(* CODESYS project PLC_Program.project

Project tree, tasks and I/O mapping:
  Device : CODESYS Control Win V3, 3S - Smart Software Solutions GmbH, order no. 305021, version 3.5.11.30
    application Application
      libraries: Standard, * (System)
      task MainTask (cyclic, interval t#20ms, priority 1) calls PLC_PRG
      task VISU_TASK (cyclic, interval 100 ms, priority 31) calls VisuElems.Visu_Prg
      program PLC_PRG [LD]
      visualisation Visualization
      Symbols
  libraries: VisuSymbols, 3.5.10.0 (System)
  text list GlobalTextList
*)

// Device/Application/PLC_PRG
PROGRAM PLC_PRG
VAR
	// TAGS DOS MÓDULOS DE ENTRADA DIGITAL E SAÍDA DIGITAL
	I0: BYTE;
	Q0: BYTE;
	// TAG DOS BLOCOS DE MEMÓRIA
	M0: BYTE;
END_VAR

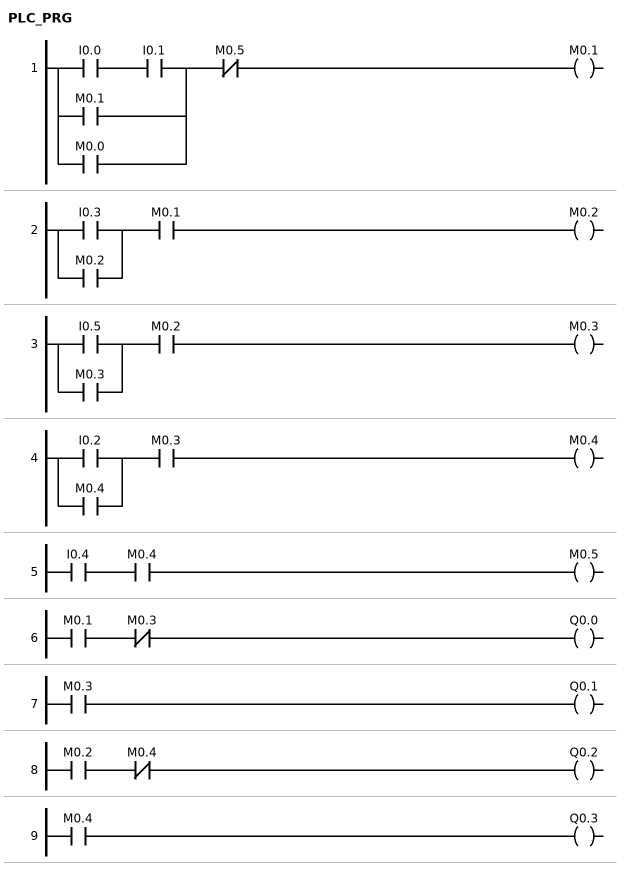
// NETWORK 1
M0.1 := (I0.0 AND I0.1 OR M0.1 OR M0.0) AND NOT M0.5;

// NETWORK 2
M0.2 := (I0.3 OR M0.2) AND M0.1;

// NETWORK 3
M0.3 := (I0.5 OR M0.3) AND M0.2;

// NETWORK 4
M0.4 := (I0.2 OR M0.4) AND M0.3;

// NETWORK 5
M0.5 := I0.4 AND M0.4;

// NETWORK 6
Q0.0 := M0.1 AND NOT M0.3;

// NETWORK 7
Q0.1 := M0.3;

// NETWORK 8
Q0.2 := M0.2 AND NOT M0.4;

// NETWORK 9
Q0.3 := M0.4;

END_PROGRAM

// Device/Application/Visualization
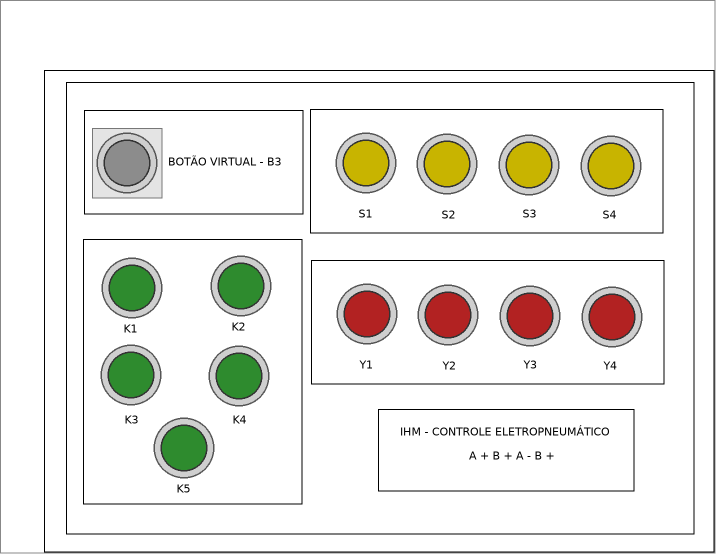
VISUALIZATION Visualization  // 716x554
    Rectangle (44,70 670x482)
    RoundedRectangle (66,82 628x452)
    RoundedRectangle (84,110 219x104)
    PushSwitch (92,128 70x70), variable: PLC_PRG.M0.0, behaviour: TOGGLE, style: Switch-PushSwitch-Gray
    Label (150,147 150x30), "BOTÃO VIRTUAL - B3"
    RoundedRectangle (310,109 353x124)
    Label (344,199 43x30), "S1"
    Lamp1 (331,128 70x70), variable: PLC_PRG.I0.2, style: Lamp-Lamp1-Yellow
    Lamp1 (412,129 70x70), variable: PLC_PRG.I0.3, style: Lamp-Lamp1-Yellow
    Lamp1 (494,130 70x70), variable: PLC_PRG.I0.4, style: Lamp-Lamp1-Yellow
    Lamp1 (576,131 70x70), variable: PLC_PRG.I0.5, style: Lamp-Lamp1-Yellow
    Label (427,200 43x30), "S2"
    Label (508,199 43x30), "S3"
    Label (588,200 43x30), "S4"
    RoundedRectangle (311,260 353x124)
    Label (345,350 43x30), "Y1"
    Lamp1 (332,279 70x70), variable: PLC_PRG.Q0.0, style: Lamp-Lamp1-Red
    Lamp1 (413,280 70x70), variable: PLC_PRG.Q0.1, style: Lamp-Lamp1-Red
    Lamp1 (495,281 70x70), variable: PLC_PRG.Q0.2, style: Lamp-Lamp1-Red
    Lamp1 (577,282 70x70), variable: PLC_PRG.Q0.3, style: Lamp-Lamp1-Red
    Label (428,351 43x30), "Y2"
    Label (509,350 43x30), "Y3"
    Label (589,351 43x30), "Y4"
    RoundedRectangle (83,239 219x265)
    Lamp1 (97,253 70x70), variable: PLC_PRG.M0.1, style: Lamp-Lamp1-Green
    Lamp1 (206,251 70x70), variable: PLC_PRG.M0.2, style: Lamp-Lamp1-Green
    Lamp1 (96,340 70x70), variable: PLC_PRG.M0.3, style: Lamp-Lamp1-Green
    Lamp1 (204,341 70x70), variable: PLC_PRG.M0.4, style: Lamp-Lamp1-Green
    Lamp1 (149,413 70x70), variable: PLC_PRG.M0.5, style: Lamp-Lamp1-Green
    Label (109,314 43x30), "K1"
    Label (217,312 43x30), "K2"
    Label (110,405 43x30), "K3"
    Label (218,405 43x30), "K4"
    Label (162,474 43x30), "K5"
    RoundedRectangle (378,409 256x82)
    Label (388,417 234x30), "IHM - CONTROLE ELETROPNEUMÁTICO"
    Label (455,441 114x30), "A + B + A - B +"
END_VISUALIZATION
